Fanuc KAREL source: kd00018.KL

-- PROVISIONAL review KL for V770-1; original PC SHA256 99ab18ad01b251e0648ee4b029e100dff03587e22df78af2decc4ace4e9b1ce5
-- Incomplete behavior may be omitted. Consult companion uncertainty JSON. Do not deploy.
PROGRAM KD00018
%NOLOCKGROUP
VAR
  I : INTEGER
  J : INTEGER
  B : BOOLEAN
  R : REAL
  S : STRING[80]
BEGIN
  -- UNRESOLVED_PC offsets 5-7; opcodes 9D,4D
  -- UNRESOLVED_PC offsets 12-16; opcodes 7F
END KD00018
